FUNCTION_BLOCK FINAL OnJsonError EXTENDS AwaitableError

END_FUNCTION_BLOCK

(* stored: Version 1.1.0.1, ProductVersion 3.1.4024.12
   POU OnJsonError: Id {04de9f32-2713-40de-b467-93156e4d7e09}, SpecialFunc None *)
